// TIA Portal V21 export
VAR_GLOBAL   // PLC tag table "K_Trends"
END_VAR
VAR_GLOBAL CONSTANT   // user constants
   K_Trend_1 : Int := 1;
   K_Trend_2 : Int := 2;
   K_Trend_3 : Int := 3;
   K_Trend_4 : Int := 4;
   K_Trend_5 : Int := 5;
   K_Trend_6 : Int := 6;
   K_Trend_7 : Int := 7;
   K_Trend_8 : Int := 8;
   K_Trend_9 : Int := 9;
   K_Trend_10 : Int := 10;
   K_Trend_11 : Int := 11;
   K_Trend_12 : Int := 12;
   K_Trend_13 : Int := 13;
   K_Trend_14 : Int := 14;
   K_Trend_15 : Int := 15;
   K_Trend_16 : Int := 16;
   K_Trend_17 : Int := 17;
   K_Trend_18 : Int := 18;
   K_Trend_19 : Int := 19;
   K_Trend_20 : Int := 20;
END_VAR
